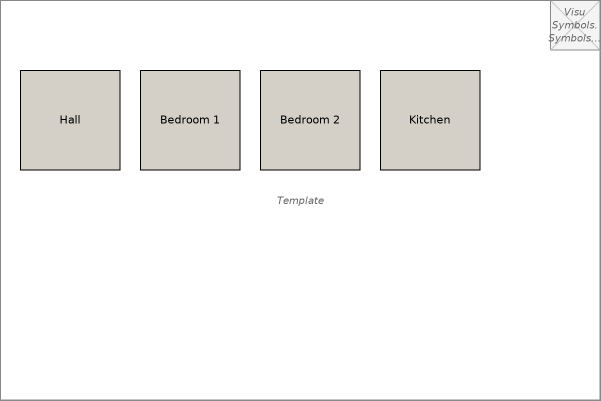
VISUALIZATION V_House  // 601x401
    Frame (0,0 601x401)
        shows Template()
    Rectangle (20,70 100x100), "Hall"
        OnMouseClick: change screen: V_Hall
    Rectangle (140,70 100x100), "Bedroom 1"
    Rectangle (260,70 100x100), "Bedroom 2"
    Rectangle (380,70 100x100), "Kitchen"
    Image (550,0 50x50), image: VisuSymbols.Symbols.Home
        OnMouseClick: change screen: V_House
END_VISUALIZATION

(* stored: Version 1.1.0.1, ProductVersion 3.1.4024.12
   Visu V_House: Id {5555882f-34ed-49b8-9325-a043c96aff3b} *)
